// Mitsubishi GX Works2 project: servo_motor_3   PLC: Q02/Q02H

PROGRAM MAIN
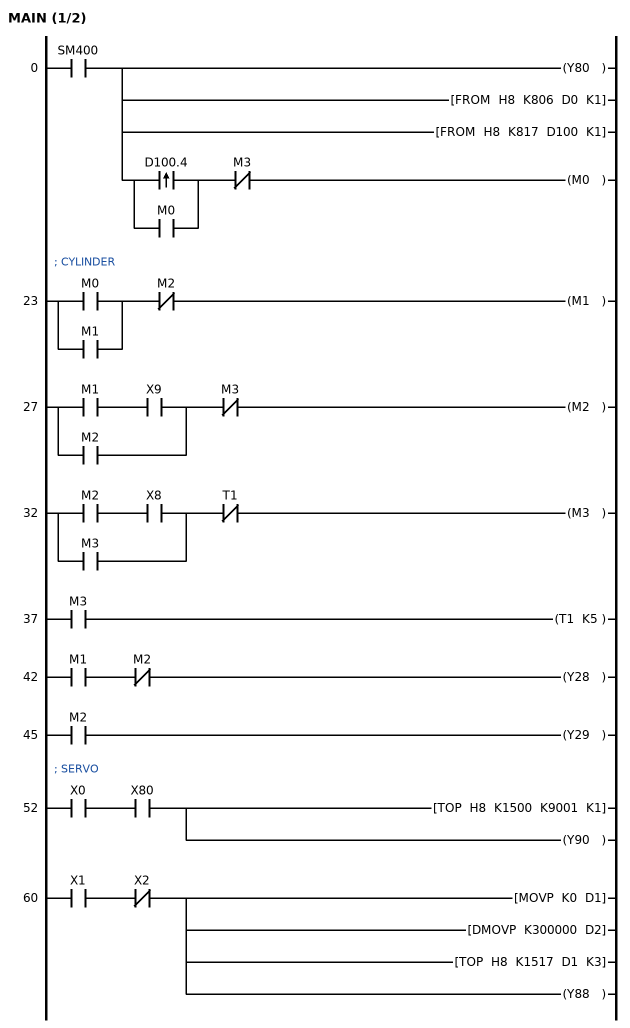
0     LD      SM400
      OUT     Y80
      FROM    H8 K806 D0 K1
      FROM    H8 K817 D100 K1
      LDP     D100.4
      OR      M0
      ANB
      ANI     M3
      OUT     M0
; CYLINDER
23    LD      M0
      OR      M1
      ANI     M2
      OUT     M1
27    LD      M1
      AND     X9
      OR      M2
      ANI     M3
      OUT     M2
32    LD      M2
      AND     X8
      OR      M3
      ANI     T1
      OUT     M3
37    LD      M3
      OUT     T1 K5
42    LD      M1
      ANI     M2
      OUT     Y28
45    LD      M2
      OUT     Y29
; SERVO
52    LD      X0
      AND     X80
      TOP     H8 K1500 K9001 K1
      OUT     Y90
60    LD      X1
      ANI     X2
      MOVP    K0 D1
      DMOVP   K300000 D2
      TOP     H8 K1517 D1 K3
      OUT     Y88
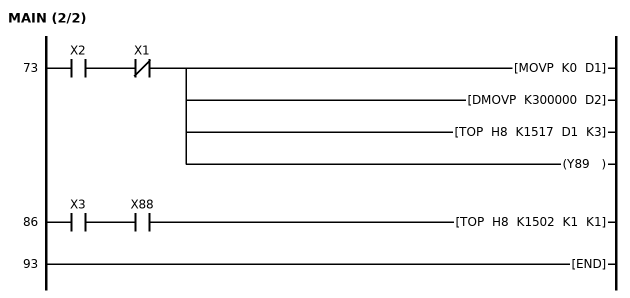
73    LD      X2
      ANI     X1
      MOVP    K0 D1
      DMOVP   K300000 D2
      TOP     H8 K1517 D1 K3
      OUT     Y89
86    LD      X3
      AND     X88
      TOP     H8 K1502 K1 K1
93    END
END_PROGRAM
